FUNCTION F_LogLA5 
VAR_INPUT
	eLogLevel		: E_LogLevel;
	sLogger			: T_MaxString;
	sMessage		: T_MaxString;
	aArg1			: ANY;
	aArg2			: ANY;
	aArg3			: ANY;
	aArg4			: ANY;
	aArg5			: ANY;
END_VAR
VAR 
	aEmptyArg		: BYTE;
END_VAR

F_LogA(
	eLogLevel,
	sLogger,
	sMessage,
	4,
	aArg1,
	aArg2,
	aArg3,
	aArg4,
	aArg5,
	aEmptyArg,
	aEmptyArg,
	aEmptyArg,
	aEmptyArg,
	aEmptyArg
);

END_FUNCTION

(* stored: Version 1.1.0.1, ProductVersion 3.1.4024.0
   POU F_LogLA5: Id {233cb8dd-cd54-4a36-8358-ee0739813912}, SpecialFunc None *)
